(* IEC 61131-3 sources: AXOpen/src/integrations/app/src/IntegrationTests/probers, 1 file *)

(* ---- ProbersTest.st ---- *)
USING AXOpen.Core;
USING AXOpen.Probers;

NAMESPACE IntegrationTests

{S7.extern=ReadWrite}
CLASS ProbersTestContext EXTENDS AxoContext
    VAR PUBLIC
        ProbeWithCounterTests : ProbeWithCounterTests;
        ProbeWithEndConditionTests : ProberWithCompletedConditionTests;
        _rootObject :   AxoObject;
    END_VAR
    METHOD PROTECTED OVERRIDE Main
        THIS.InitializeRootObject(_rootObject);
        ProbeWithCounterTests.Run(_rootObject);
        ProbeWithEndConditionTests.Run(_rootObject);
    END_METHOD
END_CLASS

{S7.extern=ReadWrite}
CLASS ProbeWithCounterTests EXTENDS AxoProberWithCounterBase
    VAR PUBLIC
        _didExecuteTestMethod : BOOL;
        _numberOfCalls : ULINT;
    END_VAR

    METHOD PROTECTED OVERRIDE Test
        _didExecuteTestMethod := TRUE;
        _numberOfCalls := _numberOfCalls + ULINT#1;
    END_METHOD
END_CLASS

{S7.extern=ReadWrite}
CLASS ProberWithCompletedConditionTests EXTENDS AxoProberWithCompletedCondition
    VAR PUBLIC
        _didExecuteTestMethod : BOOL;
        _numberOfCalls : ULINT;
    END_VAR

    METHOD PROTECTED OVERRIDE Test  : BOOL
        _didExecuteTestMethod := TRUE;
        _numberOfCalls := ULINT#123;
        Test := TRUE;
    END_METHOD
END_CLASS

END_NAMESPACE
